TYPE ST_LaudaWriteCommands_Safety :
STRUCT
	CommTimeoutViaInterface : STRING := 'OUT_SP_08_';
	ActivateSafetyMode		: STRING := 'OUT_MODE_06_';
END_STRUCT
END_TYPE

(* stored: Version 1.1.0.1, ProductVersion 3.1.4024.13
   DUT ST_LaudaWriteCommands_Safety: Id {a70ecf1d-0285-4f75-90e4-6445e094cd82} *)
